(****************************************************************************************)
(*							Beckhoff Automation Poland									*)
(*							L_TBSetBitOfWord v1.0										*)
(*									29.02.2007											*)
(*				This function sets a single bit in a value of type ”word” to “1”		*)
(*______________________________________________________________________________________*)
FUNCTION L_TBSetBitOfWord : WORD
VAR_INPUT
	wInput: WORD;
	byBitNr: BYTE;
END_VAR
VAR
END_VAR

L_TBSetBitOfWord := wInput;
CASE byBitNr OF
	0:
	L_TBSetBitOfWord.0 := TRUE;
	1:
	L_TBSetBitOfWord.1 := TRUE;
	2:
	L_TBSetBitOfWord.2 := TRUE;
	3:
	L_TBSetBitOfWord.3 := TRUE;
	4:
	L_TBSetBitOfWord.4 := TRUE;
	5:
	L_TBSetBitOfWord.5 := TRUE;
	6:
	L_TBSetBitOfWord.6 := TRUE;
	7:
	L_TBSetBitOfWord.7 := TRUE;
	8:
	L_TBSetBitOfWord.8 := TRUE;
	9:
	L_TBSetBitOfWord.9 := TRUE;
	10:
	L_TBSetBitOfWord.10 := TRUE;
	11:
	L_TBSetBitOfWord.11 := TRUE;
	12:
	L_TBSetBitOfWord.12 := TRUE;
	13:
	L_TBSetBitOfWord.13 := TRUE;
	14:
	L_TBSetBitOfWord.14 := TRUE;
	15:
	L_TBSetBitOfWord.15 := TRUE;
END_CASE

END_FUNCTION

(* stored: Version 1.1.0.1, ProductVersion 3.1.4026.13, FileIdentifier 06021c2dc290b58c6eacd351a438713ccb818f07, FileSignature 11ea332f17be5ff394df5ab793e71e71a3b6342ccd295b90768370d9b0ee270670ebd63dcee187045555a4f6422eee5d3f1ebbb04dac296a0a3afc640db868100d6898e12748f123614c72a2ad090ad01eea15e05f29fdefdd8b2750f402e53d032a785fbc13f5f8de7762bd356b380f2e1ee270be6f1b51c81416a15ebaab664c8be2d27b76455a637731975b9ee79f88e3f533a9a4752b17b05fde41829134d805d67d3bf7d611940debb18d73a29e2aa0885f098b2f74d454cf4c08f67f0c178f42b0a12667f44a64a502684607a273bee2ea8c30ea476da9f3902121b57e23edbc131c5ff2952641c76777ba689e9e4126c6286ef479e545b3406f6e2f09
   POU L_TBSetBitOfWord: Id {f6c05a83-8149-4788-bc58-f7357cf0834c}, SpecialFunc None *)
